Staubli VAL3: remGetStagePos.pgx

program remGetStagePos(string& sReturn[] (dimensions=1))
  local string sCmd
begin
  // Return the PPS status saved in the robot
  //
  logMsg("call remGetStagePos")
  sCmd="GETSTAGEPOS"
  call remGetnGlobal(nStagePos,sCmd,sReturn)
end
